TYPE ASCF_CC_OPCUACS_Writer_Temp_Bool :
STRUCT
	stReadListReturnInfo	: ARRAY [1..1] OF ST_UAReadListReturnInfo;
	Value		: BOOL		:= false;
END_STRUCT
END_TYPE

(* stored: Version 1.1.0.1, ProductVersion 3.1.4026.4
   DUT ASCF_CC_OPCUACS_Writer_Temp_Bool: Id {0da7794e-8fc4-41eb-8a8b-0f37907593a5} *)
